FUNCTION_BLOCK EM_Turning IMPLEMENTS  ITF_EM_Turning
VAR_INPUT
END_VAR
VAR_OUTPUT
END_VAR
VAR
END_VAR

END_FUNCTION_BLOCK

(* stored: Version 1.1.0.1, ProductVersion 3.1.4024.12
   POU EM_Turning: Id {eaf6caee-694c-487a-bcb2-56621ab22d66}, SpecialFunc None *)
